Staubli VAL3: recvMsgHeader.pgx

public program recvMsgHeader()
  local bool l_bFlag
begin
  // attempt to receive message prefix and header
  call recvData(siTcpIpMotion,rosGenericMsg.prefix.nData,nDataIn,l_bFlag)
  if (l_bFlag)
    call recvData(siTcpIpMotion,rosGenericMsg.header.nData,nDataIn,l_bFlag)
  endIf

  if (l_bFlag)
    // move on to state 1: decode header
    nDataInState=1
  else
    // error: reset state to 0: receive header
    nDataInState=0
  endIf


  //  // attempt to receive message header
  //  l_nBytesRecv = 0
  //  l_nIndex = 0
  //
  //  while (l_nBytesRecv < 16)
  //    l_nIndex = sioGet(siTcpIpMotion, l_nByte)
  //    if (l_nIndex == -1)
  //      if (l_nBytesRecv == 0)
  //        // 11000: client is not connected?
  //        if (nDataIn == 1)
  //          nDataIn = -1
  //        endIf
  //      else
  //        // 11000: connection lost
  //        if (nDataIn == 1)
  //          nDataIn = -1
  //        endIf
  //      endIf
  //      bValidMsgHeader = false
  //      return
  //    elseIf (l_nIndex == 1)
  //      if (l_nBytesRecv < 4)
  //        rosGenericMsg.prefix.nData[l_nBytesRecv] = l_nByte
  //      else
  //        rosGenericMsg.header.nData[l_nBytesRecv-4] = l_nByte
  //      endIf
  //      l_nBytesRecv = l_nBytesRecv + l_nIndex
  //    endIf
  //  endWhile
  //  bValidMsgHeader = true
end
